FUNCTION_BLOCK FB_ExampleDeviceSM
VAR_INPUT
	i_xMoveStarted	:	BOOL; //Connect to moving flag
	i_xMoveDone	:	BOOL; //Connect to move done flag
	i_xBeamReady	:	BOOL; //Connect to transitioneer
	i_xStopDone	:	BOOL; //Connect to MC_Stop.Done
END_VAR
VAR_OUTPUT
	q_xStartMove	:	BOOL; //Connect to MC_Absolute.Execute
	q_xStop			:	BOOL; //Connect to MC_Stop.Execute
	q_rTargetPosition	:	REAL; //Connect to MC_Absolute.Position
	q_stRequiredBeamParametersID	:	UDINT;
	q_stRequiredBeamParameters	:	ST_BeamParams; //Connect to BeamParameterTransitionManager
END_VAR
VAR_IN_OUT
	stDevice	:	ST_Device;
END_VAR
VAR
	nTargetState	:	INT;
	
	xNewReq	:	BOOL; //Set true when new target request present
	
END_VAR

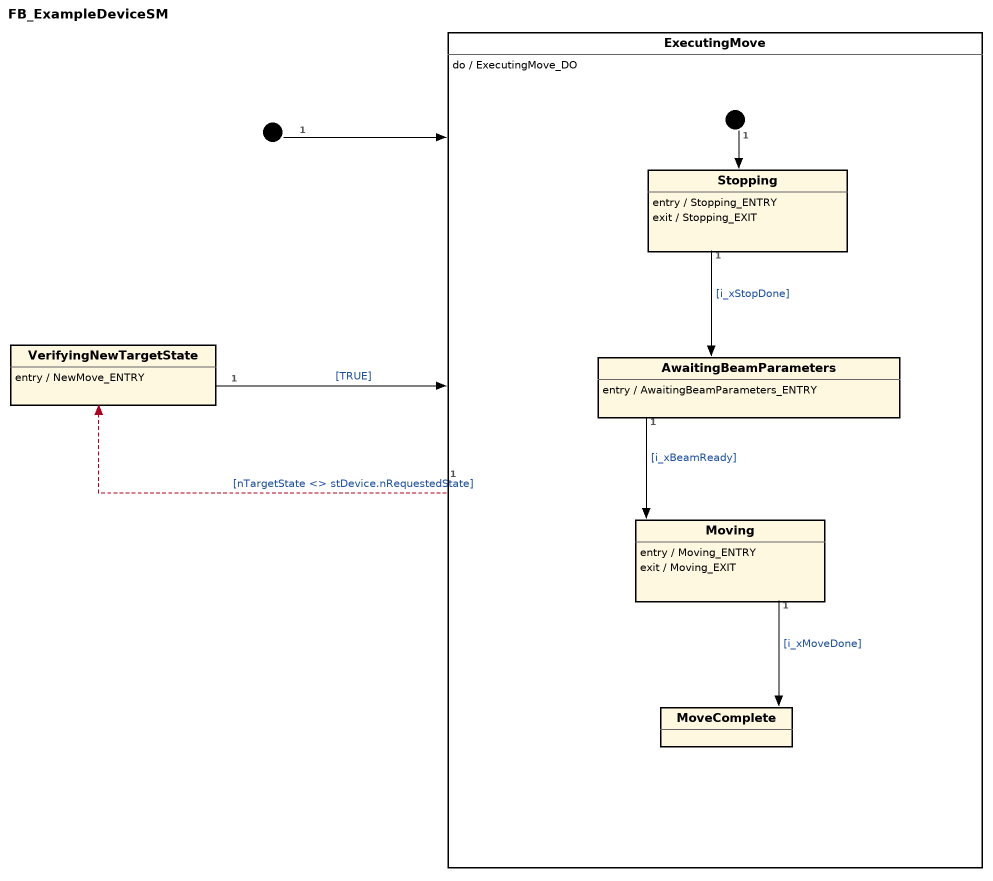
STATECHART FB_ExampleDeviceSM  // abortable
    START StartState1
    COMPOSITE STATE ExecutingMove
        do / ExecutingMove_DO
        START StartState2
        STATE Stopping
            entry / Stopping_ENTRY
            exit / Stopping_EXIT
        STATE AwaitingBeamParameters
            entry / AwaitingBeamParameters_ENTRY
        STATE Moving
            entry / Moving_ENTRY
            exit / Moving_EXIT
        STATE MoveComplete
        StartState2 -> Stopping  // priority 1, on completion
        Stopping -> AwaitingBeamParameters [i_xStopDone] // priority 1, rising edge
        AwaitingBeamParameters -> Moving [i_xBeamReady] // priority 1, rising edge
        Moving -> MoveComplete [i_xMoveDone] // priority 1, rising edge
    END_STATE
    STATE VerifyingNewTargetState
        entry / NewMove_ENTRY
    StartState1 -> ExecutingMove  // priority 1, on completion
    ExecutingMove -> VerifyingNewTargetState [nTargetState <> stDevice.nRequestedState] // priority 1, exception, rising edge
    VerifyingNewTargetState -> ExecutingMove [TRUE] // priority 1
END_STATECHART

ACTION AwaitingBeamParameters_ENTRY:
q_stRequiredBeamParameters := stDevice.astStates[nTargetState].stReqBeamParam;
q_stRequiredBeamParametersID := stDevice.astStates[nTargetState].nStateRef;
END_ACTION

ACTION ExecutingMove_DO:

END_ACTION

ACTION Moving_ENTRY:
q_xStartMove := TRUE;
q_rTargetPosition := stDevice.astStates[nTargetState].rPosition;
END_ACTION

ACTION Moving_EXIT:
q_xStartMove := FALSE;
END_ACTION

ACTION NewMove_ENTRY:

IF stDevice.nRequestedState <= PMPS_GVL_BeamParams.cnMaxStateArrayLen AND
	stDevice.nRequestedState >= 1 THEN
	nTargetState := stDevice.nRequestedState;
END_IF
END_ACTION

ACTION Stopping_ENTRY:
q_xStop	:= TRUE;
END_ACTION

ACTION Stopping_EXIT:
q_xStop := FALSE;
END_ACTION

END_FUNCTION_BLOCK

(* stored: Version 1.1.0.1, ProductVersion 3.1.4022.12
   POU FB_ExampleDeviceSM: Id {4fca12eb-f878-0f8b-0082-9204266bfe62}, SpecialFunc None
   Action AwaitingBeamParameters_ENTRY: Id {162dff85-46a9-0c88-2f29-e0c5dd18aa3c}
   Action ExecutingMove_DO: Id {3838c7d8-99b2-076e-353b-9945190676b5}
   Action Moving_ENTRY: Id {d37cd748-fdee-084f-04e4-575f7ecd1e4e}
   Action Moving_EXIT: Id {9428df2c-cfc0-0d17-11a0-bfd75af97c69}
   Action NewMove_ENTRY: Id {a217aebb-a953-088a-084d-73e66a94beed}
   Action Stopping_ENTRY: Id {8031509c-9a1a-0124-3986-403fb011568c}
   Action Stopping_EXIT: Id {ac82869e-dfe7-0a57-352b-c5a074c6fb0f} *)
